FUNCTION ServoManualMotion
VAR_INPUT
END_VAR
VAR
END_VAR

//Move to home
IF  NOT MeasuringData.AutomaticMode AND MeasuringData.MoveToHomeByManual THEN
	MAIN.AxisControl(ExecuteHomeByManual := TRUE);
ELSE
	MAIN.AxisControl(ExecuteHomeByManual := FALSE);
END_IF

//Move to bin1, bin2, bin3, bin4
IF NOT MeasuringData.AutomaticMode AND MeasuringData.MoveToBin1PositionByManual THEN
		MAIN.AxisControl(AbsolutePosition := MeasuringData.Bin1Position);
	ELSIF NOT MeasuringData.AutomaticMode AND MeasuringData.MoveToBin2PositionByManual THEN
		MAIN.AxisControl(AbsolutePosition := MeasuringData.Bin2Position);
	ELSIF NOT MeasuringData.AutomaticMode AND MeasuringData.MoveToBin3PositionByManual THEN
		MAIN.AxisControl(AbsolutePosition := MeasuringData.Bin3Position);
	ELSIF NOT MeasuringData.AutomaticMode AND MeasuringData.MoveToBin4PositionByManual THEN
		MAIN.AxisControl(AbsolutePosition := MeasuringData.Bin4Position);
	ELSE
		MAIN.AxisControl(AbsolutePosition := 0.0);
END_IF


//If one of the button is clicked on the HMI
IF (NOT MeasuringData.AutomaticMode AND MeasuringData.MoveToBin1PositionByManual) OR
	(NOT MeasuringData.AutomaticMode AND MeasuringData.MoveToBin2PositionByManual) OR
	(NOT MeasuringData.AutomaticMode AND MeasuringData.MoveToBin3PositionByManual) OR
	(NOT MeasuringData.AutomaticMode AND MeasuringData.MoveToBin4PositionByManual) THEN
	MAIN.AxisControl(ExecuteMoveAbsoluteByManual := TRUE);
ELSE
	MAIN.AxisControl(ExecuteMoveAbsoluteByManual := FALSE);
END_IF

END_FUNCTION

(* stored: Version 1.1.0.1, ProductVersion 3.1.4024.13
   POU ServoManualMotion: Id {d49eda9a-fd3f-47a2-9d2d-6548127ba3fc}, SpecialFunc None *)
